// TIA Portal V19 export
FUNCTION "EH_Promag_300_PD" : Void   // FC121, STL
TITLE = E+H_Promag_300_PD Device Process Data
{ S7_Optimized_Access := 'TRUE' }
AUTHOR : NH
FAMILY : IO_Link
NAME : EHPro300
// stored: AutoNumber false
   VAR_INPUT
      Addr : Int;   // First Byte address of 35 byte address space
      Totaliser_Mode : Byte;   // Configuration variable
   END_VAR
   VAR_OUTPUT
      Volume_Flow : Real;   // Measured value: floating point number
      Actual_Diagnostics : Int;   // Diagnostic information number
      Totaliser_Value : Real;   // Measured value: floating point number
      Device_Status_VF : Byte;   // Status Code Hex Value
      Device_Status_AD : Byte;   // Status Code Hex Value
      Device_Status_TV : Byte;   // Status Code Hex Value
   END_VAR
   VAR_IN_OUT
      Totaliser_Control : Byte;   // Control variable
   END_VAR
   VAR_TEMP
      TW_Flag : Word;
      TempInt : Int;
   END_VAR
BEGIN

NETWORK
TITLE = 
// Volume_Flow + Diagnostics
      L     #Addr;
      SLW   3;
      LAR1;

      L     ID [AR1, P#0.0];
      T     #Volume_Flow;

      L     IB [AR1, P#4.0];
      T     #Device_Status_VF;

// Actual_Diagnostics
      L     IW [AR1, P#5.0];
      T     #Actual_Diagnostics;

      L     IB [AR1, P#7.0];
      T     #Device_Status_AD;

// Totaliser_Value + Diagnostics
      L     ID [AR1, P#20.0];
      T     #Totaliser_Value;

      L     IB [AR1, P#24.0];
      T     #Device_Status_TV;

// Totaliser_Control
      L     #Totaliser_Control;
      T     QB [AR1, P#20.0];

// Totaliser_Mode
      L     #Totaliser_Mode;
      T     QB [AR1, P#21.0];





END_FUNCTION
